FUNCTION_BLOCK FB_CTD_UDINT (* counters (down-counter) *)
  (* Standard: 61131-3; Classification: counters *)
  (* Version 1.0, 2009-09-14, 4DIAC-IDE, 4DIAC-Consortium *)
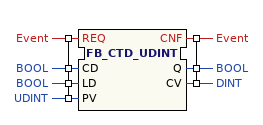
  EVENT_INPUT
    REQ WITH CD, PV, LD; (* Service Request *)
  END_EVENT
  EVENT_OUTPUT
    CNF WITH Q, CV; (* Confirmation of Requested Service *)
  END_EVENT
  VAR_INPUT
    CD : BOOL; (* Count down (Rising Edge Detection) *)
    LD : BOOL; (* Load *)
    PV : UDINT; (* Preset value *)
  END_VAR
  VAR_OUTPUT
    Q : BOOL; (* Output *)
    CV : DINT; (* Count value *)
  END_VAR
  (* Service APPLICATION/RESOURCE: counters (down-counter) *)
END_FUNCTION_BLOCK
